// TIA Portal project "Frezarka_pneumatyczna" (V14)

(* hardware
DEVICE "S7-1200 station_1"  S7-1200 Station
   slot 0: "Rack_0"  S7-1200 Rack  Rack  V1.0
   slot 1: "PLC_1"  CPU 1214C DC/DC/DC  6ES7 214-1AG40-0XB0  V4.1
   slot 2: "DI 8x24VDC_1"  6ES7 221-1BF32-0XB0  V2.0
   slot 3: "DQ 8x24VDC _1"  SM 1222 DQ8 x 24VDC  6ES7 222-1BF32-0XB0  V2.0
*)

// ===== PLC "PLC_1"  CPU 1214C DC/DC/DC =====

VAR_GLOBAL   // PLC tag table "Default tag table"
   "Clock_Byte" AT %MB50 : Byte;
   "Clock_10Hz" AT %M50.0 : Bool;
   "Clock_5Hz" AT %M50.1 : Bool;
   "Clock_2.5Hz" AT %M50.2 : Bool;
   "Clock_2Hz" AT %M50.3 : Bool;
   "Clock_1.25Hz" AT %M50.4 : Bool;
   "Clock_1Hz" AT %M50.5 : Bool;
   "Clock_0.625Hz" AT %M50.6 : Bool;
   "Clock_0.5Hz" AT %M50.7 : Bool;
   "Magazyn_pusty" AT %M0.0 : Bool;
   "System_Byte" AT %MB51 : Byte;
   "FirstScan" AT %M51.0 : Bool;
   "DiagStatusUpdate" AT %M51.1 : Bool;
   "AlwaysTRUE" AT %M51.2 : Bool;
   "AlwaysFALSE" AT %M51.3 : Bool;
END_VAR

VAR_GLOBAL   // PLC tag table "Wejscia cyfrowe"
   "Start" AT %I0.0 : Bool;
   "Stop" AT %I0.1 : Bool;
   "Stop_awaryjny" AT %I0.2 : Bool;
   "Praca_auto" AT %I0.3 : Bool;
   "Praca_jeden_cykl" AT %I0.4 : Bool;
   "Krancowka_S1-" AT %I0.5 : Bool;
   "Krancowka_S1+" AT %I0.6 : Bool;
   "Krancowka_S2-" AT %I0.7 : Bool;
   "Krancowka_S2+" AT %I1.0 : Bool;
   "Krancowka_S3-" AT %I1.1 : Bool;
   "Krancowka_S3+" AT %I1.2 : Bool;
   "Krancowka_S4-" AT %I1.3 : Bool;
   "Krancowka_S4+" AT %I1.4 : Bool;
   "Magazyn" AT %I1.5 : Bool;
   "Potwierdzenie_wrzeciono" AT %I2.0 : Bool;
   "Start_silownik1" AT %I2.1 : Bool;
   "Start_silownik2" AT %I2.2 : Bool;
   "Start_silownik3" AT %I2.3 : Bool;
   "Start_silownik4" AT %I2.4 : Bool;
   "Start_wrzeciono" AT %I2.5 : Bool;
   "Stop_wrzeciono" AT %I2.6 : Bool;
END_VAR

VAR_GLOBAL   // PLC tag table "Wyjscia cyfrowe"
   "Silownik1" AT %Q0.0 : Bool;
   "Silownik2" AT %Q0.1 : Bool;
   "Silownik3" AT %Q0.2 : Bool;
   "Silownik4" AT %Q0.3 : Bool;
   "Wrzeciono" AT %Q0.4 : Bool;
   "Silnik_trojkat" AT %Q0.5 : Bool;
   "Silnik_gwiazda" AT %Q0.6 : Bool;
   "Lampka_awaria" AT %Q0.7 : Bool;
   "Lampka_start" AT %Q1.0 : Bool;
   "Lampka_praca_auto" AT %Q2.0 : Bool;
   "Lampka_praca_reczna" AT %Q2.1 : Bool;
   "Wysuwanie_silownika1" AT %Q2.2 : Bool;
   "Wysuwanie_silownika2" AT %Q2.3 : Bool;
   "Wysuwanie_silownika3" AT %Q2.4 : Bool;
   "Wysuwanie_silownika4" AT %Q2.5 : Bool;
END_VAR

DATA_BLOCK "Zmienne_do_automatu"   // DB1
{ S7_Optimized_Access := 'TRUE' }
VERSION : 0.1
   VAR
      Q1 : Bool;
      Q2 : Bool;
      Q3 : Bool;
      Q4 : Bool;
      Q5 : Bool;
   END_VAR
BEGIN
END_DATA_BLOCK

DATA_BLOCK "Automat_sterujacy_DB"   // DB2
{ S7_Optimized_Access := 'TRUE' }
VERSION : 0.1
// stored: InstanceOfName Automat_sterujacy_auto
"Automat_sterujacy_auto"
BEGIN
END_DATA_BLOCK

DATA_BLOCK "Sprawdzenie_magazynu_DB"   // DB4
{ S7_Optimized_Access := 'TRUE' }
VERSION : 0.1
// stored: InstanceOfName Sprawdzenie_magazynu
"Sprawdzenie_magazynu"
BEGIN
END_DATA_BLOCK

// folder: System blocks/Program resources

DATA_BLOCK "Timer_magazyn"   // DB3
{ S7_Optimized_Access := 'TRUE' }
AUTHOR : Simatic
FAMILY : IEC
NAME : IEC_TMR
VERSION : 1.0
// stored: InstanceOfName IEC_TIMER
"IEC_TIMER"
BEGIN
END_DATA_BLOCK

DATA_BLOCK "IEC_Timer_0_DB"   // DB5
{ S7_Optimized_Access := 'TRUE' }
AUTHOR : Simatic
FAMILY : IEC
NAME : IEC_TMR
VERSION : 1.0
// stored: InstanceOfName IEC_TIMER
"IEC_TIMER"
BEGIN
END_DATA_BLOCK

DATA_BLOCK "IEC_Timer_0_DB_1"   // DB6
{ S7_Optimized_Access := 'TRUE' }
AUTHOR : Simatic
FAMILY : IEC
NAME : IEC_TMR
VERSION : 1.0
// stored: InstanceOfName IEC_TIMER
"IEC_TIMER"
BEGIN
END_DATA_BLOCK

DATA_BLOCK "IEC_Counter_0_DB"   // DB7
{ S7_Optimized_Access := 'TRUE' }
AUTHOR : Simatic
FAMILY : IEC
NAME : CNTR
VERSION : 1.0
// stored: InstanceOfName IEC_COUNTER
"IEC_COUNTER"
BEGIN
END_DATA_BLOCK

// folder: (top level)

FUNCTION_BLOCK "Automat_sterujacy_auto"   // FB1, LAD
{ S7_Optimized_Access := 'TRUE' }
VERSION : 0.1
// WEJSCIE W STAN1
   VAR_INPUT
      Stop : Bool;
      Stop_awaryjny : Bool;
      Magazyn : Bool;
      Tryb_pracy_auto : Bool;
   END_VAR
   VAR_OUTPUT
      Silownik1 : Bool;
      Silownik2 : Bool;
      Silownik3 : Bool;
      Silownik4 : Bool;
      Wrzeciono : Bool;
   END_VAR
   VAR
      S0 : Bool;   // STAN0
      S1 : Bool;   // STAN1
      S2 : Bool;   // STAN2
      S3 : Bool;   // STAN3
      S4 : Bool;   // STAN4
      S5 : Bool;   // STAN5
      S6 : Bool;   // STAN6
      S7 : Bool;   // STAN7
      S8 : Bool;   // STAN8
      Podtrzymaj_stop : Bool;
      Podtrzymaj_tryb : Bool;
      TMP : Bool;
   END_VAR
   VAR_TEMP   // added for the SCL form of the ladder/FBD networks
      _w1 : Bool;
   END_VAR
BEGIN

REGION Network 1: STAN1
   // RESET WSZYSTKICH STANÓW PODCZAS STOPU AWARYJNEGO LUB PUSTEGO MAGAZYNU
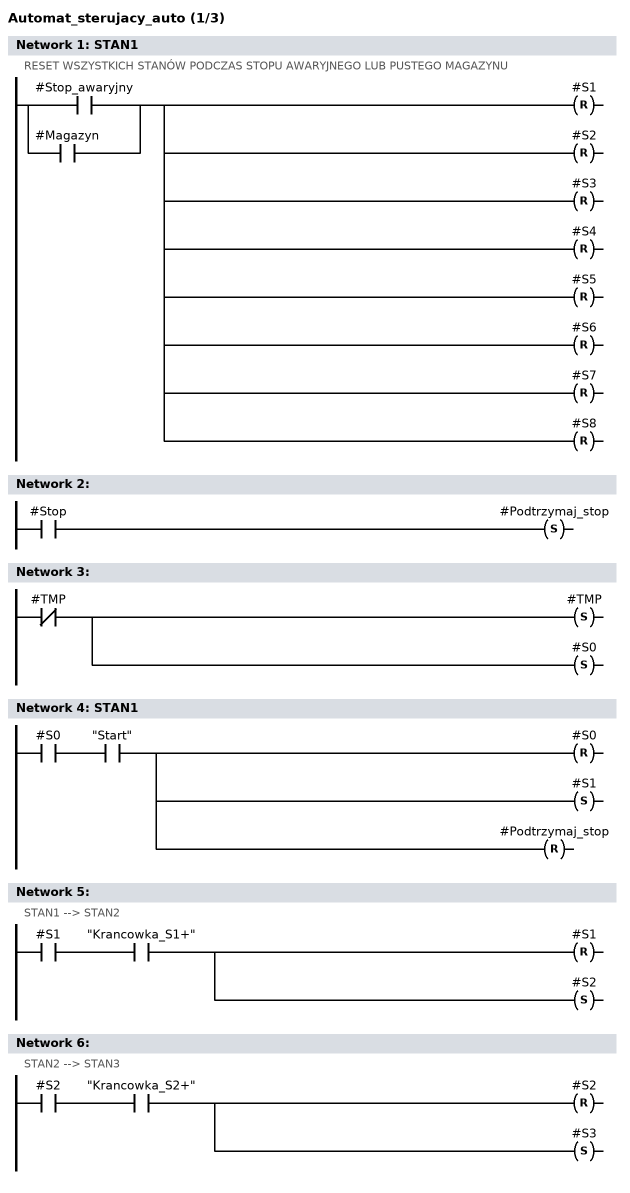
   RUNG wire#powerrail
      Contact( #Stop_awaryjny )
      wire#w1
      R_Coil( #S1 )
   END_RUNG
   RUNG wire#powerrail
      Contact( #Magazyn )
   END_RUNG wire#w1
   RUNG wire#w1
      R_Coil( #S2 )
   END_RUNG
   RUNG wire#w1
      R_Coil( #S3 )
   END_RUNG
   RUNG wire#w1
      R_Coil( #S4 )
   END_RUNG
   RUNG wire#w1
      R_Coil( #S5 )
   END_RUNG
   RUNG wire#w1
      R_Coil( #S6 )
   END_RUNG
   RUNG wire#w1
      R_Coil( #S7 )
   END_RUNG
   RUNG wire#w1
      R_Coil( #S8 )
   END_RUNG
   // the same network as SCL:
   IF #Stop_awaryjny OR #Magazyn THEN
       #S1 := FALSE;
       #S2 := FALSE;
       #S3 := FALSE;
       #S4 := FALSE;
       #S5 := FALSE;
       #S6 := FALSE;
       #S7 := FALSE;
       #S8 := FALSE;
   END_IF;
END_REGION

REGION Network 2
   RUNG wire#powerrail
      Contact( #Stop )
      S_Coil( #Podtrzymaj_stop )
   END_RUNG
   // the same network as SCL:
   IF #Stop THEN #Podtrzymaj_stop := TRUE; END_IF;
END_REGION

REGION Network 3
   RUNG wire#powerrail
      I_Contact( #TMP )
      wire#w1
      S_Coil( #TMP )
   END_RUNG
   RUNG wire#w1
      S_Coil( #S0 )
   END_RUNG
   // the same network as SCL:
   #_w1 := NOT #TMP;
   IF #_w1 THEN
       #TMP := TRUE;
       #S0 := TRUE;
   END_IF;
END_REGION

REGION Network 4: STAN1
   RUNG wire#powerrail
      Contact( #S0 )
      Contact( "Start" )
      wire#w1
      R_Coil( #S0 )
   END_RUNG
   RUNG wire#w1
      S_Coil( #S1 )
   END_RUNG
   RUNG wire#w1
      R_Coil( #Podtrzymaj_stop )
   END_RUNG
   // the same network as SCL:
   #_w1 := #S0 AND "Start";
   IF #_w1 THEN
       #S0 := FALSE;
       #S1 := TRUE;
       #Podtrzymaj_stop := FALSE;
   END_IF;
END_REGION

REGION Network 5
   // STAN1 --> STAN2
   RUNG wire#powerrail
      Contact( #S1 )
      Contact( "Krancowka_S1+" )
      wire#w1
      R_Coil( #S1 )
   END_RUNG
   RUNG wire#w1
      S_Coil( #S2 )
   END_RUNG
   // the same network as SCL:
   #_w1 := #S1 AND "Krancowka_S1+";
   IF #_w1 THEN
       #S1 := FALSE;
       #S2 := TRUE;
   END_IF;
END_REGION

REGION Network 6
   // STAN2 --> STAN3
   RUNG wire#powerrail
      Contact( #S2 )
      Contact( "Krancowka_S2+" )
      wire#w1
      R_Coil( #S2 )
   END_RUNG
   RUNG wire#w1
      S_Coil( #S3 )
   END_RUNG
   // the same network as SCL:
   #_w1 := #S2 AND "Krancowka_S2+";
   IF #_w1 THEN
       #S2 := FALSE;
       #S3 := TRUE;
   END_IF;
END_REGION

REGION Network 7
   // STAN3 --> STAN4
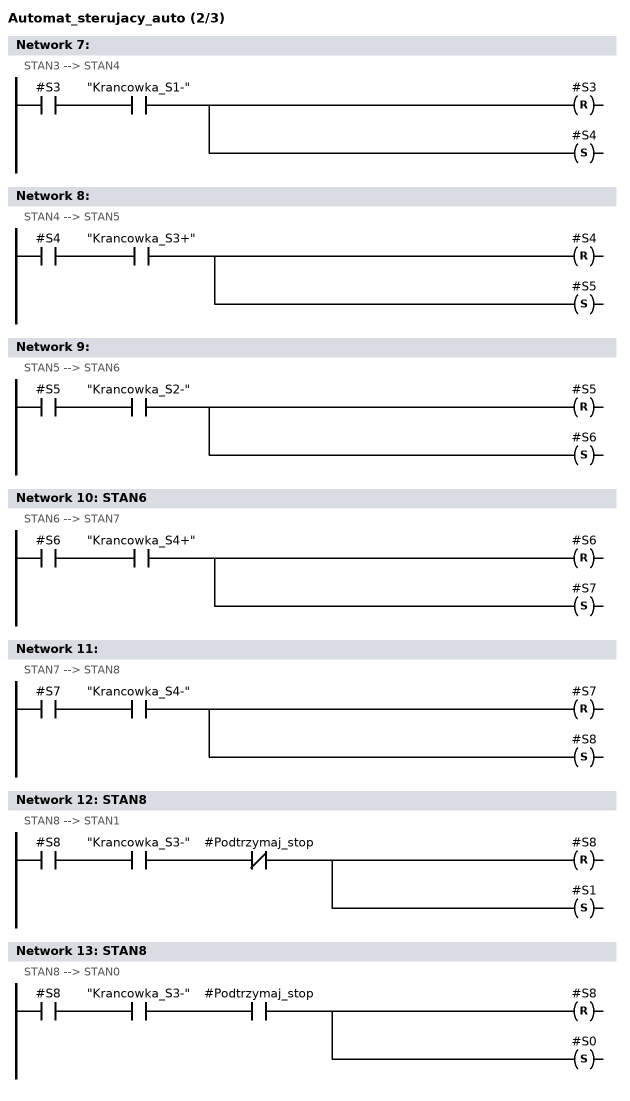
   RUNG wire#powerrail
      Contact( #S3 )
      Contact( "Krancowka_S1-" )
      wire#w1
      R_Coil( #S3 )
   END_RUNG
   RUNG wire#w1
      S_Coil( #S4 )
   END_RUNG
   // the same network as SCL:
   #_w1 := #S3 AND "Krancowka_S1-";
   IF #_w1 THEN
       #S3 := FALSE;
       #S4 := TRUE;
   END_IF;
END_REGION

REGION Network 8
   // STAN4 --> STAN5
   RUNG wire#powerrail
      Contact( #S4 )
      Contact( "Krancowka_S3+" )
      wire#w1
      R_Coil( #S4 )
   END_RUNG
   RUNG wire#w1
      S_Coil( #S5 )
   END_RUNG
   // the same network as SCL:
   #_w1 := #S4 AND "Krancowka_S3+";
   IF #_w1 THEN
       #S4 := FALSE;
       #S5 := TRUE;
   END_IF;
END_REGION

REGION Network 9
   // STAN5 --> STAN6
   RUNG wire#powerrail
      Contact( #S5 )
      Contact( "Krancowka_S2-" )
      wire#w1
      R_Coil( #S5 )
   END_RUNG
   RUNG wire#w1
      S_Coil( #S6 )
   END_RUNG
   // the same network as SCL:
   #_w1 := #S5 AND "Krancowka_S2-";
   IF #_w1 THEN
       #S5 := FALSE;
       #S6 := TRUE;
   END_IF;
END_REGION

REGION Network 10: STAN6
   // STAN6 --> STAN7
   RUNG wire#powerrail
      Contact( #S6 )
      Contact( "Krancowka_S4+" )
      wire#w1
      R_Coil( #S6 )
   END_RUNG
   RUNG wire#w1
      S_Coil( #S7 )
   END_RUNG
   // the same network as SCL:
   #_w1 := #S6 AND "Krancowka_S4+";
   IF #_w1 THEN
       #S6 := FALSE;
       #S7 := TRUE;
   END_IF;
END_REGION

REGION Network 11
   // STAN7 --> STAN8
   RUNG wire#powerrail
      Contact( #S7 )
      Contact( "Krancowka_S4-" )
      wire#w1
      R_Coil( #S7 )
   END_RUNG
   RUNG wire#w1
      S_Coil( #S8 )
   END_RUNG
   // the same network as SCL:
   #_w1 := #S7 AND "Krancowka_S4-";
   IF #_w1 THEN
       #S7 := FALSE;
       #S8 := TRUE;
   END_IF;
END_REGION

REGION Network 12: STAN8
   // STAN8 --> STAN1
   RUNG wire#powerrail
      Contact( #S8 )
      Contact( "Krancowka_S3-" )
      I_Contact( #Podtrzymaj_stop )
      wire#w1
      R_Coil( #S8 )
   END_RUNG
   RUNG wire#w1
      S_Coil( #S1 )
   END_RUNG
   // the same network as SCL:
   #_w1 := #S8 AND "Krancowka_S3-" AND NOT #Podtrzymaj_stop;
   IF #_w1 THEN
       #S8 := FALSE;
       #S1 := TRUE;
   END_IF;
END_REGION

REGION Network 13: STAN8
   // STAN8 --> STAN0
   RUNG wire#powerrail
      Contact( #S8 )
      Contact( "Krancowka_S3-" )
      Contact( #Podtrzymaj_stop )
      wire#w1
      R_Coil( #S8 )
   END_RUNG
   RUNG wire#w1
      S_Coil( #S0 )
   END_RUNG
   // the same network as SCL:
   #_w1 := #S8 AND "Krancowka_S3-" AND #Podtrzymaj_stop;
   IF #_w1 THEN
       #S8 := FALSE;
       #S0 := TRUE;
   END_IF;
END_REGION

REGION Network 14
   // WYJSCIE SILOWNIK1
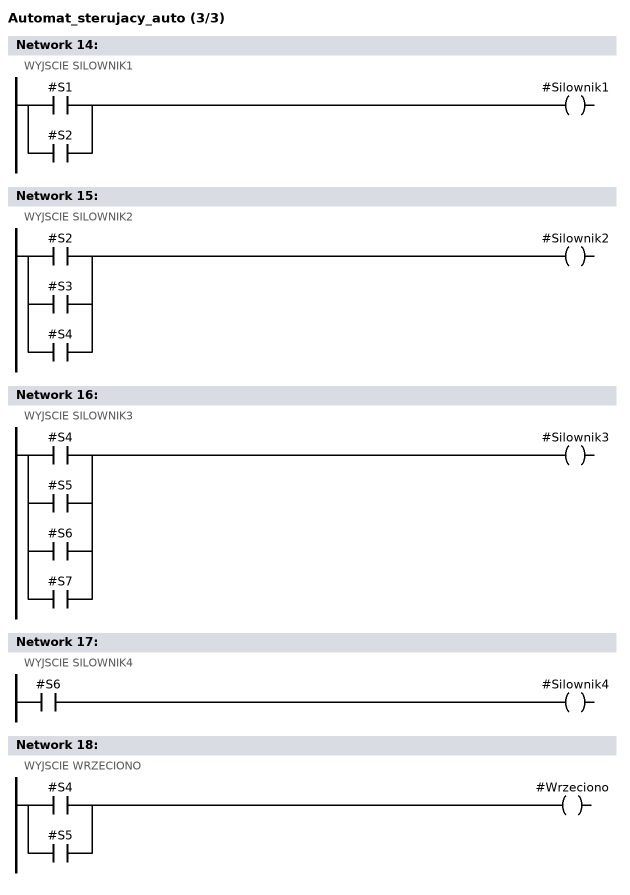
   RUNG wire#powerrail
      Contact( #S1 )
      wire#w1
      Coil( #Silownik1 )
   END_RUNG
   RUNG wire#powerrail
      Contact( #S2 )
   END_RUNG wire#w1
   // the same network as SCL:
   #Silownik1 := #S1 OR #S2;
END_REGION

REGION Network 15
   // WYJSCIE SILOWNIK2
   RUNG wire#powerrail
      Contact( #S2 )
      wire#w1
      Coil( #Silownik2 )
   END_RUNG
   RUNG wire#powerrail
      Contact( #S3 )
   END_RUNG wire#w1
   RUNG wire#powerrail
      Contact( #S4 )
   END_RUNG wire#w1
   // the same network as SCL:
   #Silownik2 := #S2 OR #S3 OR #S4;
END_REGION

REGION Network 16
   // WYJSCIE SILOWNIK3
   RUNG wire#powerrail
      Contact( #S4 )
      wire#w1
      Coil( #Silownik3 )
   END_RUNG
   RUNG wire#powerrail
      Contact( #S5 )
   END_RUNG wire#w1
   RUNG wire#powerrail
      Contact( #S6 )
   END_RUNG wire#w1
   RUNG wire#powerrail
      Contact( #S7 )
   END_RUNG wire#w1
   // the same network as SCL:
   #Silownik3 := #S4 OR #S5 OR #S6 OR #S7;
END_REGION

REGION Network 17
   // WYJSCIE SILOWNIK4
   RUNG wire#powerrail
      Contact( #S6 )
      Coil( #Silownik4 )
   END_RUNG
   // the same network as SCL:
   #Silownik4 := #S6;
END_REGION

REGION Network 18
   // WYJSCIE WRZECIONO
   RUNG wire#powerrail
      Contact( #S4 )
      wire#w1
      Coil( #Wrzeciono )
   END_RUNG
   RUNG wire#powerrail
      Contact( #S5 )
   END_RUNG wire#w1
   // the same network as SCL:
   #Wrzeciono := #S4 OR #S5;
END_REGION
END_FUNCTION_BLOCK

FUNCTION_BLOCK "Automat_sterujacy_jeden_cykl"   // FB1, LAD
{ S7_Optimized_Access := 'TRUE' }
VERSION : 0.1
// WEJSCIE W STAN1
   VAR_INPUT
      Stop : Bool;
      Stop_awaryjny : Bool;
      Magazyn : Bool;
      Tryb_pracy_auto : Bool;
   END_VAR
   VAR_OUTPUT
      Silownik1 : Bool;
      Silownik2 : Bool;
      Silownik3 : Bool;
      Silownik4 : Bool;
      Wrzeciono : Bool;
   END_VAR
   VAR
      S0 : Bool;   // STAN0
      S1 : Bool;   // STAN1
      S2 : Bool;   // STAN2
      S3 : Bool;   // STAN3
      S4 : Bool;   // STAN4
      S5 : Bool;   // STAN5
      S6 : Bool;   // STAN6
      S7 : Bool;   // STAN7
      S8 : Bool;   // STAN8
      Podtrzymaj_stop : Bool;
      Podtrzymaj_tryb : Bool;
      TMP : Bool;
   END_VAR
   VAR_TEMP   // added for the SCL form of the ladder/FBD networks
      _w1 : Bool;
   END_VAR
BEGIN

REGION Network 1: STAN1
   // RESET WSZYSTKICH STANÓW PODCZAS STOPU AWARYJNEGO LUB PUSTEGO MAGAZYNU
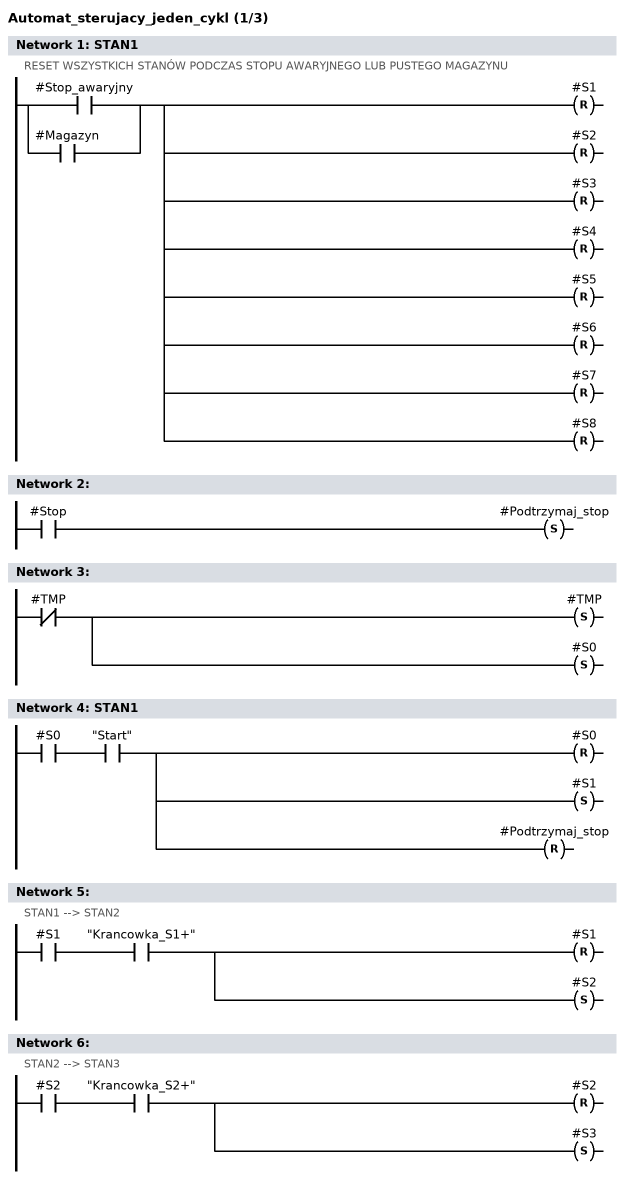
   RUNG wire#powerrail
      Contact( #Stop_awaryjny )
      wire#w1
      R_Coil( #S1 )
   END_RUNG
   RUNG wire#powerrail
      Contact( #Magazyn )
   END_RUNG wire#w1
   RUNG wire#w1
      R_Coil( #S2 )
   END_RUNG
   RUNG wire#w1
      R_Coil( #S3 )
   END_RUNG
   RUNG wire#w1
      R_Coil( #S4 )
   END_RUNG
   RUNG wire#w1
      R_Coil( #S5 )
   END_RUNG
   RUNG wire#w1
      R_Coil( #S6 )
   END_RUNG
   RUNG wire#w1
      R_Coil( #S7 )
   END_RUNG
   RUNG wire#w1
      R_Coil( #S8 )
   END_RUNG
   // the same network as SCL:
   IF #Stop_awaryjny OR #Magazyn THEN
       #S1 := FALSE;
       #S2 := FALSE;
       #S3 := FALSE;
       #S4 := FALSE;
       #S5 := FALSE;
       #S6 := FALSE;
       #S7 := FALSE;
       #S8 := FALSE;
   END_IF;
END_REGION

REGION Network 2
   RUNG wire#powerrail
      Contact( #Stop )
      S_Coil( #Podtrzymaj_stop )
   END_RUNG
   // the same network as SCL:
   IF #Stop THEN #Podtrzymaj_stop := TRUE; END_IF;
END_REGION

REGION Network 3
   RUNG wire#powerrail
      I_Contact( #TMP )
      wire#w1
      S_Coil( #TMP )
   END_RUNG
   RUNG wire#w1
      S_Coil( #S0 )
   END_RUNG
   // the same network as SCL:
   #_w1 := NOT #TMP;
   IF #_w1 THEN
       #TMP := TRUE;
       #S0 := TRUE;
   END_IF;
END_REGION

REGION Network 4: STAN1
   RUNG wire#powerrail
      Contact( #S0 )
      Contact( "Start" )
      wire#w1
      R_Coil( #S0 )
   END_RUNG
   RUNG wire#w1
      S_Coil( #S1 )
   END_RUNG
   RUNG wire#w1
      R_Coil( #Podtrzymaj_stop )
   END_RUNG
   // the same network as SCL:
   #_w1 := #S0 AND "Start";
   IF #_w1 THEN
       #S0 := FALSE;
       #S1 := TRUE;
       #Podtrzymaj_stop := FALSE;
   END_IF;
END_REGION

REGION Network 5
   // STAN1 --> STAN2
   RUNG wire#powerrail
      Contact( #S1 )
      Contact( "Krancowka_S1+" )
      wire#w1
      R_Coil( #S1 )
   END_RUNG
   RUNG wire#w1
      S_Coil( #S2 )
   END_RUNG
   // the same network as SCL:
   #_w1 := #S1 AND "Krancowka_S1+";
   IF #_w1 THEN
       #S1 := FALSE;
       #S2 := TRUE;
   END_IF;
END_REGION

REGION Network 6
   // STAN2 --> STAN3
   RUNG wire#powerrail
      Contact( #S2 )
      Contact( "Krancowka_S2+" )
      wire#w1
      R_Coil( #S2 )
   END_RUNG
   RUNG wire#w1
      S_Coil( #S3 )
   END_RUNG
   // the same network as SCL:
   #_w1 := #S2 AND "Krancowka_S2+";
   IF #_w1 THEN
       #S2 := FALSE;
       #S3 := TRUE;
   END_IF;
END_REGION

REGION Network 7
   // STAN3 --> STAN4
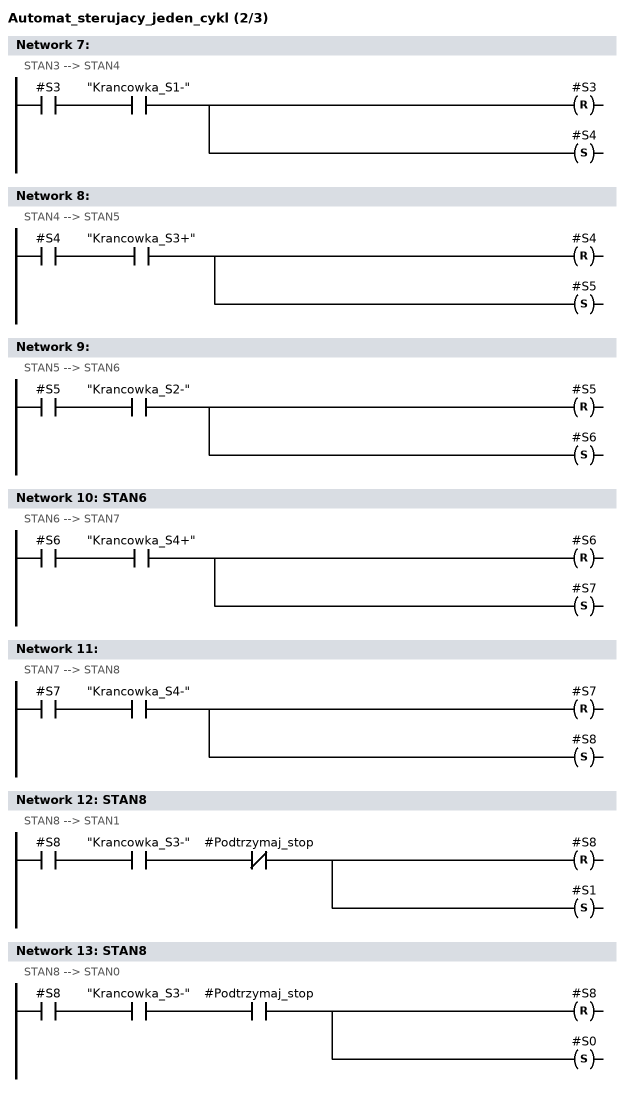
   RUNG wire#powerrail
      Contact( #S3 )
      Contact( "Krancowka_S1-" )
      wire#w1
      R_Coil( #S3 )
   END_RUNG
   RUNG wire#w1
      S_Coil( #S4 )
   END_RUNG
   // the same network as SCL:
   #_w1 := #S3 AND "Krancowka_S1-";
   IF #_w1 THEN
       #S3 := FALSE;
       #S4 := TRUE;
   END_IF;
END_REGION

REGION Network 8
   // STAN4 --> STAN5
   RUNG wire#powerrail
      Contact( #S4 )
      Contact( "Krancowka_S3+" )
      wire#w1
      R_Coil( #S4 )
   END_RUNG
   RUNG wire#w1
      S_Coil( #S5 )
   END_RUNG
   // the same network as SCL:
   #_w1 := #S4 AND "Krancowka_S3+";
   IF #_w1 THEN
       #S4 := FALSE;
       #S5 := TRUE;
   END_IF;
END_REGION

REGION Network 9
   // STAN5 --> STAN6
   RUNG wire#powerrail
      Contact( #S5 )
      Contact( "Krancowka_S2-" )
      wire#w1
      R_Coil( #S5 )
   END_RUNG
   RUNG wire#w1
      S_Coil( #S6 )
   END_RUNG
   // the same network as SCL:
   #_w1 := #S5 AND "Krancowka_S2-";
   IF #_w1 THEN
       #S5 := FALSE;
       #S6 := TRUE;
   END_IF;
END_REGION

REGION Network 10: STAN6
   // STAN6 --> STAN7
   RUNG wire#powerrail
      Contact( #S6 )
      Contact( "Krancowka_S4+" )
      wire#w1
      R_Coil( #S6 )
   END_RUNG
   RUNG wire#w1
      S_Coil( #S7 )
   END_RUNG
   // the same network as SCL:
   #_w1 := #S6 AND "Krancowka_S4+";
   IF #_w1 THEN
       #S6 := FALSE;
       #S7 := TRUE;
   END_IF;
END_REGION

REGION Network 11
   // STAN7 --> STAN8
   RUNG wire#powerrail
      Contact( #S7 )
      Contact( "Krancowka_S4-" )
      wire#w1
      R_Coil( #S7 )
   END_RUNG
   RUNG wire#w1
      S_Coil( #S8 )
   END_RUNG
   // the same network as SCL:
   #_w1 := #S7 AND "Krancowka_S4-";
   IF #_w1 THEN
       #S7 := FALSE;
       #S8 := TRUE;
   END_IF;
END_REGION

REGION Network 12: STAN8
   // STAN8 --> STAN1
   RUNG wire#powerrail
      Contact( #S8 )
      Contact( "Krancowka_S3-" )
      I_Contact( #Podtrzymaj_stop )
      wire#w1
      R_Coil( #S8 )
   END_RUNG
   RUNG wire#w1
      S_Coil( #S1 )
   END_RUNG
   // the same network as SCL:
   #_w1 := #S8 AND "Krancowka_S3-" AND NOT #Podtrzymaj_stop;
   IF #_w1 THEN
       #S8 := FALSE;
       #S1 := TRUE;
   END_IF;
END_REGION

REGION Network 13: STAN8
   // STAN8 --> STAN0
   RUNG wire#powerrail
      Contact( #S8 )
      Contact( "Krancowka_S3-" )
      Contact( #Podtrzymaj_stop )
      wire#w1
      R_Coil( #S8 )
   END_RUNG
   RUNG wire#w1
      S_Coil( #S0 )
   END_RUNG
   // the same network as SCL:
   #_w1 := #S8 AND "Krancowka_S3-" AND #Podtrzymaj_stop;
   IF #_w1 THEN
       #S8 := FALSE;
       #S0 := TRUE;
   END_IF;
END_REGION

REGION Network 14
   // WYJSCIE SILOWNIK1
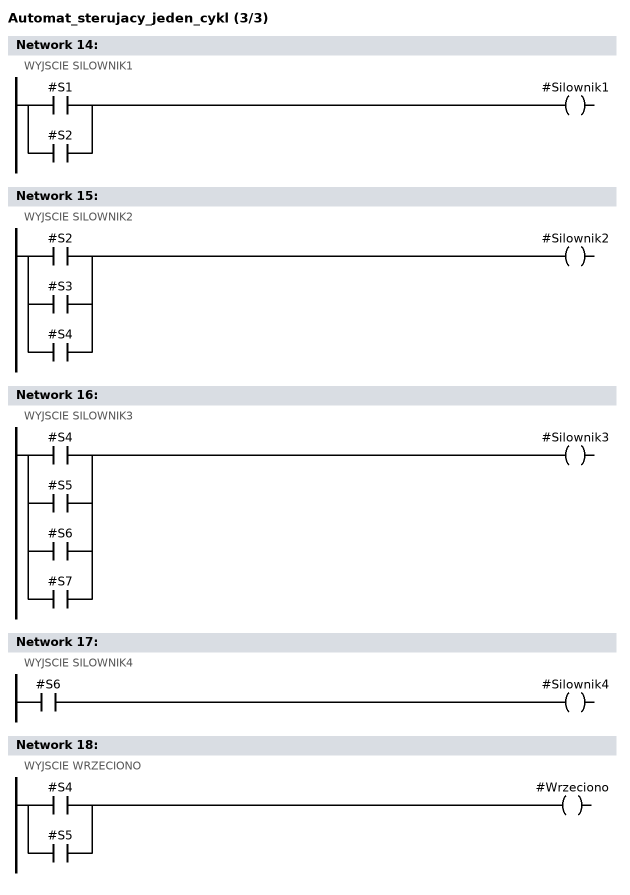
   RUNG wire#powerrail
      Contact( #S1 )
      wire#w1
      Coil( #Silownik1 )
   END_RUNG
   RUNG wire#powerrail
      Contact( #S2 )
   END_RUNG wire#w1
   // the same network as SCL:
   #Silownik1 := #S1 OR #S2;
END_REGION

REGION Network 15
   // WYJSCIE SILOWNIK2
   RUNG wire#powerrail
      Contact( #S2 )
      wire#w1
      Coil( #Silownik2 )
   END_RUNG
   RUNG wire#powerrail
      Contact( #S3 )
   END_RUNG wire#w1
   RUNG wire#powerrail
      Contact( #S4 )
   END_RUNG wire#w1
   // the same network as SCL:
   #Silownik2 := #S2 OR #S3 OR #S4;
END_REGION

REGION Network 16
   // WYJSCIE SILOWNIK3
   RUNG wire#powerrail
      Contact( #S4 )
      wire#w1
      Coil( #Silownik3 )
   END_RUNG
   RUNG wire#powerrail
      Contact( #S5 )
   END_RUNG wire#w1
   RUNG wire#powerrail
      Contact( #S6 )
   END_RUNG wire#w1
   RUNG wire#powerrail
      Contact( #S7 )
   END_RUNG wire#w1
   // the same network as SCL:
   #Silownik3 := #S4 OR #S5 OR #S6 OR #S7;
END_REGION

REGION Network 17
   // WYJSCIE SILOWNIK4
   RUNG wire#powerrail
      Contact( #S6 )
      Coil( #Silownik4 )
   END_RUNG
   // the same network as SCL:
   #Silownik4 := #S6;
END_REGION

REGION Network 18
   // WYJSCIE WRZECIONO
   RUNG wire#powerrail
      Contact( #S4 )
      wire#w1
      Coil( #Wrzeciono )
   END_RUNG
   RUNG wire#powerrail
      Contact( #S5 )
   END_RUNG wire#w1
   // the same network as SCL:
   #Wrzeciono := #S4 OR #S5;
END_REGION
END_FUNCTION_BLOCK

FUNCTION_BLOCK "Automat_sterujacy_reczne"   // FB1, LAD
{ S7_Optimized_Access := 'TRUE' }
VERSION : 0.1
// WEJSCIE W STAN1
   VAR_INPUT
      Stop : Bool;
      Stop_awaryjny : Bool;
      Magazyn : Bool;
      Tryb_pracy_auto : Bool;
   END_VAR
   VAR_OUTPUT
      Silownik1 : Bool;
      Silownik2 : Bool;
      Silownik3 : Bool;
      Silownik4 : Bool;
      Wrzeciono : Bool;
   END_VAR
   VAR
      S0 : Bool;   // STAN0
      S1 : Bool;   // STAN1
      S2 : Bool;   // STAN2
      S3 : Bool;   // STAN3
      S4 : Bool;   // STAN4
      S5 : Bool;   // STAN5
      S6 : Bool;   // STAN6
      S7 : Bool;   // STAN7
      S8 : Bool;   // STAN8
      Podtrzymaj_stop : Bool;
      Podtrzymaj_tryb : Bool;
      TMP : Bool;
   END_VAR
   VAR_TEMP   // added for the SCL form of the ladder/FBD networks
      _w1 : Bool;
   END_VAR
BEGIN

REGION Network 1: STAN1
   // RESET WSZYSTKICH STANÓW PODCZAS STOPU AWARYJNEGO LUB PUSTEGO MAGAZYNU
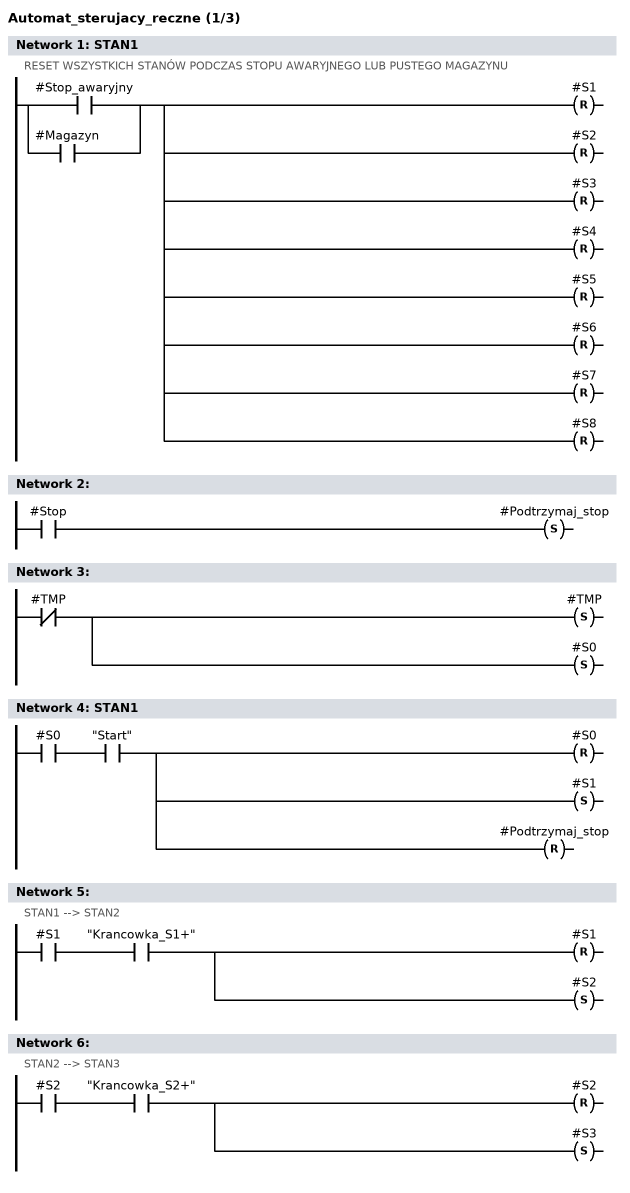
   RUNG wire#powerrail
      Contact( #Stop_awaryjny )
      wire#w1
      R_Coil( #S1 )
   END_RUNG
   RUNG wire#powerrail
      Contact( #Magazyn )
   END_RUNG wire#w1
   RUNG wire#w1
      R_Coil( #S2 )
   END_RUNG
   RUNG wire#w1
      R_Coil( #S3 )
   END_RUNG
   RUNG wire#w1
      R_Coil( #S4 )
   END_RUNG
   RUNG wire#w1
      R_Coil( #S5 )
   END_RUNG
   RUNG wire#w1
      R_Coil( #S6 )
   END_RUNG
   RUNG wire#w1
      R_Coil( #S7 )
   END_RUNG
   RUNG wire#w1
      R_Coil( #S8 )
   END_RUNG
   // the same network as SCL:
   IF #Stop_awaryjny OR #Magazyn THEN
       #S1 := FALSE;
       #S2 := FALSE;
       #S3 := FALSE;
       #S4 := FALSE;
       #S5 := FALSE;
       #S6 := FALSE;
       #S7 := FALSE;
       #S8 := FALSE;
   END_IF;
END_REGION

REGION Network 2
   RUNG wire#powerrail
      Contact( #Stop )
      S_Coil( #Podtrzymaj_stop )
   END_RUNG
   // the same network as SCL:
   IF #Stop THEN #Podtrzymaj_stop := TRUE; END_IF;
END_REGION

REGION Network 3
   RUNG wire#powerrail
      I_Contact( #TMP )
      wire#w1
      S_Coil( #TMP )
   END_RUNG
   RUNG wire#w1
      S_Coil( #S0 )
   END_RUNG
   // the same network as SCL:
   #_w1 := NOT #TMP;
   IF #_w1 THEN
       #TMP := TRUE;
       #S0 := TRUE;
   END_IF;
END_REGION

REGION Network 4: STAN1
   RUNG wire#powerrail
      Contact( #S0 )
      Contact( "Start" )
      wire#w1
      R_Coil( #S0 )
   END_RUNG
   RUNG wire#w1
      S_Coil( #S1 )
   END_RUNG
   RUNG wire#w1
      R_Coil( #Podtrzymaj_stop )
   END_RUNG
   // the same network as SCL:
   #_w1 := #S0 AND "Start";
   IF #_w1 THEN
       #S0 := FALSE;
       #S1 := TRUE;
       #Podtrzymaj_stop := FALSE;
   END_IF;
END_REGION

REGION Network 5
   // STAN1 --> STAN2
   RUNG wire#powerrail
      Contact( #S1 )
      Contact( "Krancowka_S1+" )
      wire#w1
      R_Coil( #S1 )
   END_RUNG
   RUNG wire#w1
      S_Coil( #S2 )
   END_RUNG
   // the same network as SCL:
   #_w1 := #S1 AND "Krancowka_S1+";
   IF #_w1 THEN
       #S1 := FALSE;
       #S2 := TRUE;
   END_IF;
END_REGION

REGION Network 6
   // STAN2 --> STAN3
   RUNG wire#powerrail
      Contact( #S2 )
      Contact( "Krancowka_S2+" )
      wire#w1
      R_Coil( #S2 )
   END_RUNG
   RUNG wire#w1
      S_Coil( #S3 )
   END_RUNG
   // the same network as SCL:
   #_w1 := #S2 AND "Krancowka_S2+";
   IF #_w1 THEN
       #S2 := FALSE;
       #S3 := TRUE;
   END_IF;
END_REGION

REGION Network 7
   // STAN3 --> STAN4
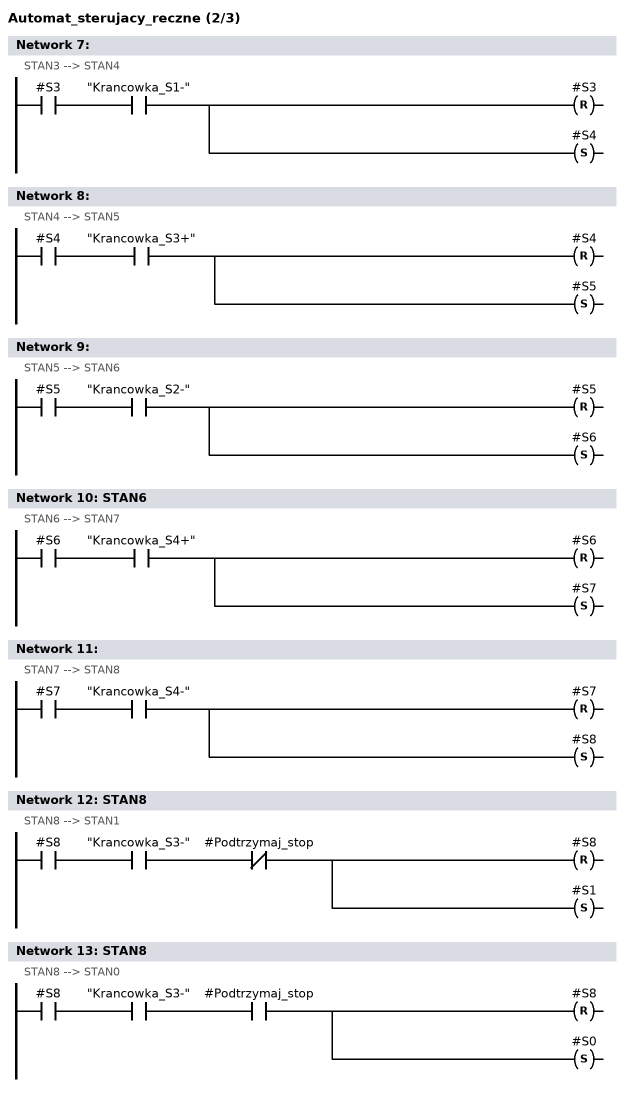
   RUNG wire#powerrail
      Contact( #S3 )
      Contact( "Krancowka_S1-" )
      wire#w1
      R_Coil( #S3 )
   END_RUNG
   RUNG wire#w1
      S_Coil( #S4 )
   END_RUNG
   // the same network as SCL:
   #_w1 := #S3 AND "Krancowka_S1-";
   IF #_w1 THEN
       #S3 := FALSE;
       #S4 := TRUE;
   END_IF;
END_REGION

REGION Network 8
   // STAN4 --> STAN5
   RUNG wire#powerrail
      Contact( #S4 )
      Contact( "Krancowka_S3+" )
      wire#w1
      R_Coil( #S4 )
   END_RUNG
   RUNG wire#w1
      S_Coil( #S5 )
   END_RUNG
   // the same network as SCL:
   #_w1 := #S4 AND "Krancowka_S3+";
   IF #_w1 THEN
       #S4 := FALSE;
       #S5 := TRUE;
   END_IF;
END_REGION

REGION Network 9
   // STAN5 --> STAN6
   RUNG wire#powerrail
      Contact( #S5 )
      Contact( "Krancowka_S2-" )
      wire#w1
      R_Coil( #S5 )
   END_RUNG
   RUNG wire#w1
      S_Coil( #S6 )
   END_RUNG
   // the same network as SCL:
   #_w1 := #S5 AND "Krancowka_S2-";
   IF #_w1 THEN
       #S5 := FALSE;
       #S6 := TRUE;
   END_IF;
END_REGION

REGION Network 10: STAN6
   // STAN6 --> STAN7
   RUNG wire#powerrail
      Contact( #S6 )
      Contact( "Krancowka_S4+" )
      wire#w1
      R_Coil( #S6 )
   END_RUNG
   RUNG wire#w1
      S_Coil( #S7 )
   END_RUNG
   // the same network as SCL:
   #_w1 := #S6 AND "Krancowka_S4+";
   IF #_w1 THEN
       #S6 := FALSE;
       #S7 := TRUE;
   END_IF;
END_REGION

REGION Network 11
   // STAN7 --> STAN8
   RUNG wire#powerrail
      Contact( #S7 )
      Contact( "Krancowka_S4-" )
      wire#w1
      R_Coil( #S7 )
   END_RUNG
   RUNG wire#w1
      S_Coil( #S8 )
   END_RUNG
   // the same network as SCL:
   #_w1 := #S7 AND "Krancowka_S4-";
   IF #_w1 THEN
       #S7 := FALSE;
       #S8 := TRUE;
   END_IF;
END_REGION

REGION Network 12: STAN8
   // STAN8 --> STAN1
   RUNG wire#powerrail
      Contact( #S8 )
      Contact( "Krancowka_S3-" )
      I_Contact( #Podtrzymaj_stop )
      wire#w1
      R_Coil( #S8 )
   END_RUNG
   RUNG wire#w1
      S_Coil( #S1 )
   END_RUNG
   // the same network as SCL:
   #_w1 := #S8 AND "Krancowka_S3-" AND NOT #Podtrzymaj_stop;
   IF #_w1 THEN
       #S8 := FALSE;
       #S1 := TRUE;
   END_IF;
END_REGION

REGION Network 13: STAN8
   // STAN8 --> STAN0
   RUNG wire#powerrail
      Contact( #S8 )
      Contact( "Krancowka_S3-" )
      Contact( #Podtrzymaj_stop )
      wire#w1
      R_Coil( #S8 )
   END_RUNG
   RUNG wire#w1
      S_Coil( #S0 )
   END_RUNG
   // the same network as SCL:
   #_w1 := #S8 AND "Krancowka_S3-" AND #Podtrzymaj_stop;
   IF #_w1 THEN
       #S8 := FALSE;
       #S0 := TRUE;
   END_IF;
END_REGION

REGION Network 14
   // WYJSCIE SILOWNIK1
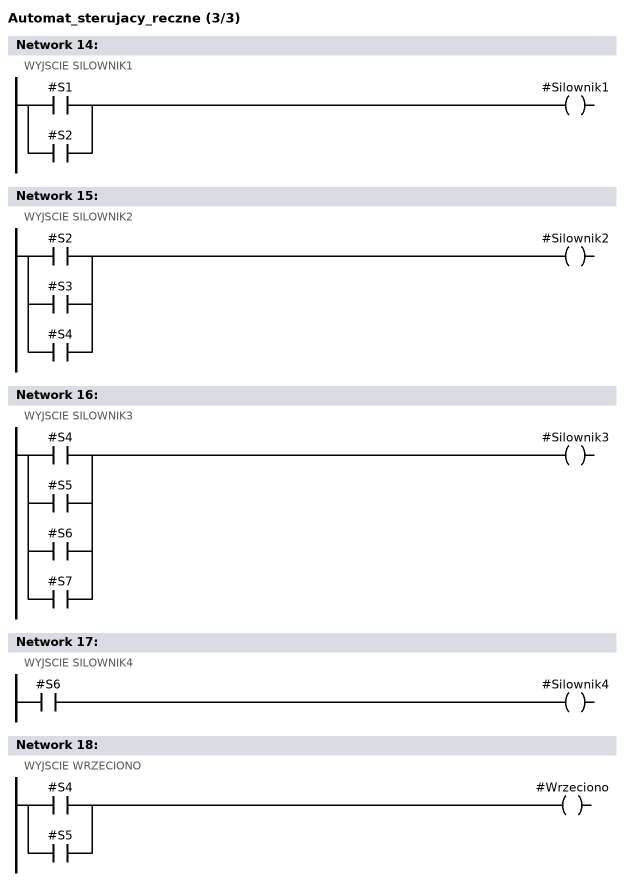
   RUNG wire#powerrail
      Contact( #S1 )
      wire#w1
      Coil( #Silownik1 )
   END_RUNG
   RUNG wire#powerrail
      Contact( #S2 )
   END_RUNG wire#w1
   // the same network as SCL:
   #Silownik1 := #S1 OR #S2;
END_REGION

REGION Network 15
   // WYJSCIE SILOWNIK2
   RUNG wire#powerrail
      Contact( #S2 )
      wire#w1
      Coil( #Silownik2 )
   END_RUNG
   RUNG wire#powerrail
      Contact( #S3 )
   END_RUNG wire#w1
   RUNG wire#powerrail
      Contact( #S4 )
   END_RUNG wire#w1
   // the same network as SCL:
   #Silownik2 := #S2 OR #S3 OR #S4;
END_REGION

REGION Network 16
   // WYJSCIE SILOWNIK3
   RUNG wire#powerrail
      Contact( #S4 )
      wire#w1
      Coil( #Silownik3 )
   END_RUNG
   RUNG wire#powerrail
      Contact( #S5 )
   END_RUNG wire#w1
   RUNG wire#powerrail
      Contact( #S6 )
   END_RUNG wire#w1
   RUNG wire#powerrail
      Contact( #S7 )
   END_RUNG wire#w1
   // the same network as SCL:
   #Silownik3 := #S4 OR #S5 OR #S6 OR #S7;
END_REGION

REGION Network 17
   // WYJSCIE SILOWNIK4
   RUNG wire#powerrail
      Contact( #S6 )
      Coil( #Silownik4 )
   END_RUNG
   // the same network as SCL:
   #Silownik4 := #S6;
END_REGION

REGION Network 18
   // WYJSCIE WRZECIONO
   RUNG wire#powerrail
      Contact( #S4 )
      wire#w1
      Coil( #Wrzeciono )
   END_RUNG
   RUNG wire#powerrail
      Contact( #S5 )
   END_RUNG wire#w1
   // the same network as SCL:
   #Wrzeciono := #S4 OR #S5;
END_REGION
END_FUNCTION_BLOCK

FUNCTION_BLOCK "Sprawdzenie_magazynu"   // FB2, LAD
{ S7_Optimized_Access := 'TRUE' }
VERSION : 0.1
   VAR_OUTPUT
      Magazyn_pusty : Bool;
   END_VAR
BEGIN

REGION Network 1
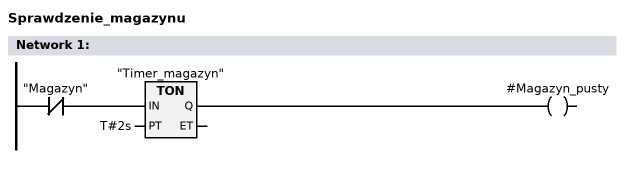
   "Timer_magazyn".TON(IN := NOT "Magazyn", PT := T#2s);
   #Magazyn_pusty := "Timer_magazyn".Q;
END_REGION
END_FUNCTION_BLOCK

ORGANIZATION_BLOCK "Main"   // OB1, LAD, ProgramCycle
TITLE = "Main Program Sweep (Cycle)"
{ S7_Optimized_Access := 'TRUE' }
VERSION : 0.1
   VAR_INPUT
      Initial_Call : Bool;   // Initial call of this OB
      Remanence : Bool;   // =True, if remanent data are available
   END_VAR
BEGIN

REGION Network 1
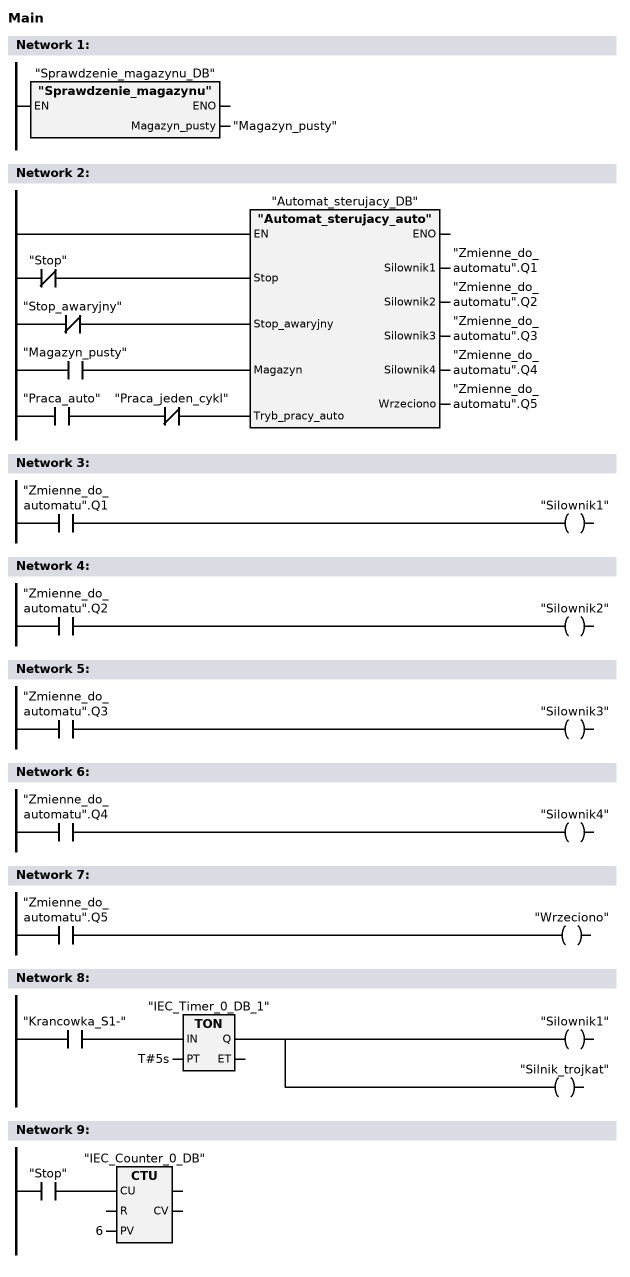
   RUNG wire#powerrail
      "Sprawdzenie_magazynu_DB"(Magazyn_pusty => "Magazyn_pusty")
   END_RUNG
   // the same network as SCL:
   "Sprawdzenie_magazynu_DB"(Magazyn_pusty => "Magazyn_pusty");   // "Sprawdzenie_magazynu"
END_REGION

REGION Network 2
   RUNG wire#powerrail
      "Automat_sterujacy_DB"(Stop := wire#w1, Stop_awaryjny := wire#w2, Magazyn := wire#w3, Tryb_pracy_auto := wire#w4, Silownik1 => "Zmienne_do_automatu".Q1, Silownik2 => "Zmienne_do_automatu".Q2, Silownik3 => "Zmienne_do_automatu".Q3, Silownik4 => "Zmienne_do_automatu".Q4, Wrzeciono => "Zmienne_do_automatu".Q5)
   END_RUNG
   RUNG wire#powerrail
      I_Contact( "Stop" )
   END_RUNG wire#w1
   RUNG wire#powerrail
      I_Contact( "Stop_awaryjny" )
   END_RUNG wire#w2
   RUNG wire#powerrail
      Contact( "Magazyn_pusty" )
   END_RUNG wire#w3
   RUNG wire#powerrail
      Contact( "Praca_auto" )
      I_Contact( "Praca_jeden_cykl" )
   END_RUNG wire#w4
   // the same network as SCL:
   "Automat_sterujacy_DB"(Stop := NOT "Stop",   // "Automat_sterujacy_auto"
                          Stop_awaryjny := NOT "Stop_awaryjny",
                          Magazyn := "Magazyn_pusty",
                          Tryb_pracy_auto := "Praca_auto" AND NOT "Praca_jeden_cykl",
                          Silownik1 => "Zmienne_do_automatu".Q1,
                          Silownik2 => "Zmienne_do_automatu".Q2,
                          Silownik3 => "Zmienne_do_automatu".Q3,
                          Silownik4 => "Zmienne_do_automatu".Q4,
                          Wrzeciono => "Zmienne_do_automatu".Q5);
END_REGION

REGION Network 3
   RUNG wire#powerrail
      Contact( "Zmienne_do_automatu".Q1 )
      Coil( "Silownik1" )
   END_RUNG
   // the same network as SCL:
   "Silownik1" := "Zmienne_do_automatu".Q1;
END_REGION

REGION Network 4
   RUNG wire#powerrail
      Contact( "Zmienne_do_automatu".Q2 )
      Coil( "Silownik2" )
   END_RUNG
   // the same network as SCL:
   "Silownik2" := "Zmienne_do_automatu".Q2;
END_REGION

REGION Network 5
   RUNG wire#powerrail
      Contact( "Zmienne_do_automatu".Q3 )
      Coil( "Silownik3" )
   END_RUNG
   // the same network as SCL:
   "Silownik3" := "Zmienne_do_automatu".Q3;
END_REGION

REGION Network 6
   RUNG wire#powerrail
      Contact( "Zmienne_do_automatu".Q4 )
      Coil( "Silownik4" )
   END_RUNG
   // the same network as SCL:
   "Silownik4" := "Zmienne_do_automatu".Q4;
END_REGION

REGION Network 7
   RUNG wire#powerrail
      Contact( "Zmienne_do_automatu".Q5 )
      Coil( "Wrzeciono" )
   END_RUNG
   // the same network as SCL:
   "Wrzeciono" := "Zmienne_do_automatu".Q5;
END_REGION

REGION Network 8
   "IEC_Timer_0_DB_1".TON(IN := "Krancowka_S1-", PT := T#5s);
   "Silownik1" := "IEC_Timer_0_DB_1".Q;
   "Silnik_trojkat" := "IEC_Timer_0_DB_1".Q;
END_REGION

REGION Network 9
   "IEC_Counter_0_DB".CTU(CU := "Stop", PV := 6);
END_REGION
END_ORGANIZATION_BLOCK

ORGANIZATION_BLOCK "Time delay interrupt"   // OB20, LAD, TimeDelayInterrupt
{ S7_Optimized_Access := 'TRUE' }
VERSION : 0.1
   VAR_INPUT
      Sign : Word;   // Identifier input (SIGN) passed to triggering call of SRT_DINT
   END_VAR
BEGIN
END_ORGANIZATION_BLOCK

ORGANIZATION_BLOCK "Cyclic interrupt"   // OB30, LAD, CyclicInterrupt
{ S7_Optimized_Access := 'TRUE' }
VERSION : 0.1
   VAR_INPUT
      Initial_Call : Bool;   // Initial call of this OB
      Event_Count : Int;   // Events discarded
   END_VAR
BEGIN
END_ORGANIZATION_BLOCK

ORGANIZATION_BLOCK "Hardware interrupt"   // OB40, LAD, HWProcessInterrupt
{ S7_Optimized_Access := 'TRUE' }
VERSION : 0.1
   VAR_INPUT
      LADDR : Hw_Io;   // Hardware identifier
      USI : Word;   // User structure identifier
      IChannel : USInt;   // Interrupt channel number
      EventType : Byte;   // EventType
   END_VAR
BEGIN
END_ORGANIZATION_BLOCK

ORGANIZATION_BLOCK "Startup"   // OB100, LAD, Startup
TITLE = "Complete Restart"
{ S7_Optimized_Access := 'TRUE' }
VERSION : 0.1
   VAR_INPUT
      LostRetentive : Bool;   // True if retentive data are lost
      LostRTC : Bool;   // True if date and time are lost
   END_VAR
BEGIN
END_ORGANIZATION_BLOCK